% RSLogix 500 project DOOR_CON.RSS, saved by version 8.30.00.16 %
PROJECT "DOOR_CON"    % processor: Bul.1763 MicroLogix 1100 Series B %

PROGRAM FILES
  LAD 2   3 rungs

DATA FILES
  O0 OUTPUT  4 elements
  I1 INPUT  6 elements
  S2 STATUS  66 elements
  B3 BINARY  1 elements
  T4 TIMER  1 elements
  C5 COUNTER  1 elements
  R6 CONTROL  1 elements
  N7 INTEGER  1 elements
  F8 FLOAT  1 elements

LADDER 2
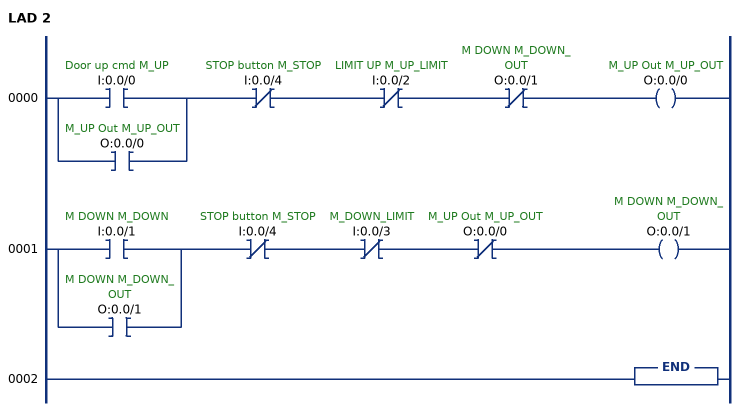
% Rung: 0 %  % edit flag set %
SOR BST XIC I:0.0/0 NXB XIC O:0.0/0 BND XIO I:0.0/4 XIO I:0.0/2 XIO O:0.0/1 OTE O:0.0/0 EOR
%   I:0.0/0  M_UP  "Door up cmd" %
%   O:0.0/0  M_UP_OUT  "M_UP Out" %
%   I:0.0/4  M_STOP  "STOP button" %
%   I:0.0/2  M_UP_LIMIT  "LIMIT UP" %
%   O:0.0/1  M_DOWN_OUT  "M DOWN" %
% Rung: 1 %  % edit flag set %
SOR BST XIC I:0.0/1 NXB XIC O:0.0/1 BND XIO I:0.0/4 XIO I:0.0/3 XIO O:0.0/0 OTE O:0.0/1 EOR
%   I:0.0/1  M_DOWN  "M DOWN" %
%   O:0.0/1  M_DOWN_OUT  "M DOWN" %
%   I:0.0/4  M_STOP  "STOP button" %
%   I:0.0/3  M_DOWN_LIMIT %
%   O:0.0/0  M_UP_OUT  "M_UP Out" %
% Rung: 2 %
SOR END EOR
